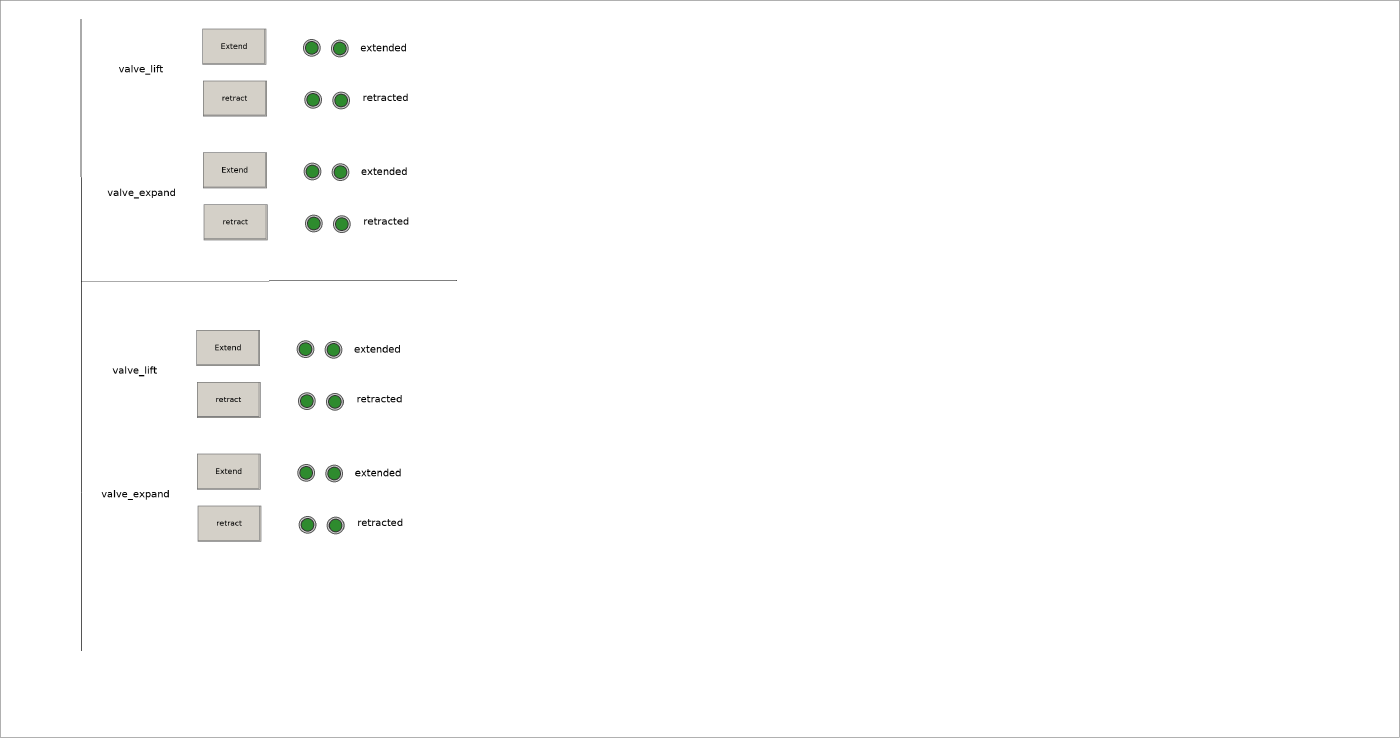
VISUALIZATION v_IO_fixtureClamp  // 2048x1080
    Line (118,28) (119,952)
    Label (126,88 160x26), "valve_lift"
    Button (296,42 93x52), "Extend", colour toggle: G_IO.arDO[55].Ch[10]
        OnMouseDown: execute { G_IO.arDO[55].Ch[10] := TRUE; G_IO.arDO[55].Ch[11] := FALSE; }
    Button (297,118 93x52), "retract", colour toggle: G_IO.arDO[55].Ch[11]
        OnMouseDown: execute { G_IO.arDO[55].Ch[10] := FALSE; G_IO.arDO[55].Ch[11] := TRUE; }
    Lamp1 (441,55 30x30), variable: G_IO.arDI[77].Ch[0], style: Lamp-Lamp1-Green
    Lamp1 (443,131 30x30), variable: G_IO.arDI[77].Ch[1], style: Lamp-Lamp1-Green
    Label (495,57 132x26), "extended"
    Label (498,130 132x26), "retracted"
    Lamp1 (482,56 30x30), variable: G_IO.arDI[77].Ch[2], style: Lamp-Lamp1-Green
    Lamp1 (484,132 30x30), variable: G_IO.arDI[77].Ch[3], style: Lamp-Lamp1-Green
    Label (127,269 160x26), "valve_expand"
    Button (297,223 93x52), "Extend", colour toggle: G_IO.arDO[55].Ch[12]
        OnMouseDown: execute { G_IO.arDO[55].Ch[12] := TRUE; G_IO.arDO[55].Ch[13] := FALSE; }
    Button (298,299 93x52), "retract", colour toggle: G_IO.arDO[55].Ch[13]
        OnMouseDown: execute { G_IO.arDO[55].Ch[12] := FALSE; G_IO.arDO[55].Ch[13] := TRUE; }
    Lamp1 (442,236 30x30), variable: G_IO.arDI[77].Ch[4], style: Lamp-Lamp1-Green
    Lamp1 (444,312 30x30), variable: G_IO.arDI[77].Ch[5], style: Lamp-Lamp1-Green
    Label (496,238 132x26), "extended"
    Label (499,311 132x26), "retracted"
    Lamp1 (483,237 30x30), variable: G_IO.arDI[77].Ch[6], style: Lamp-Lamp1-Green
    Lamp1 (485,313 30x30), variable: G_IO.arDI[77].Ch[7], style: Lamp-Lamp1-Green
    Label (117,529 160x26), "valve_lift"
    Button (287,483 93x52), "Extend", colour toggle: G_IO.arDO[59].Ch[10]
        OnMouseDown: execute { G_IO.arDO[59].Ch[10] := TRUE; G_IO.arDO[59].Ch[11] := FALSE; }
    Button (288,559 93x52), "retract", colour toggle: G_IO.arDO[59].Ch[11]
        OnMouseDown: execute { G_IO.arDO[59].Ch[10] := FALSE; G_IO.arDO[59].Ch[11] := TRUE; }
    Lamp1 (432,496 30x30), variable: G_IO.arDI[78].Ch[0], style: Lamp-Lamp1-Green
    Lamp1 (434,572 30x30), variable: G_IO.arDI[78].Ch[1], style: Lamp-Lamp1-Green
    Label (486,498 132x26), "extended"
    Label (489,571 132x26), "retracted"
    Lamp1 (473,497 30x30), variable: G_IO.arDI[78].Ch[2], style: Lamp-Lamp1-Green
    Lamp1 (475,573 30x30), variable: G_IO.arDI[78].Ch[3], style: Lamp-Lamp1-Green
    Label (118,710 160x26), "valve_expand"
    Button (288,664 93x52), "Extend", colour toggle: G_IO.arDO[59].Ch[12]
        OnMouseDown: execute { G_IO.arDO[59].Ch[12] := TRUE; G_IO.arDO[59].Ch[13] := FALSE; }
    Button (289,740 93x52), "retract", colour toggle: G_IO.arDO[59].Ch[13]
        OnMouseDown: execute { G_IO.arDO[59].Ch[12] := FALSE; G_IO.arDO[59].Ch[13] := TRUE; }
    Lamp1 (433,677 30x30), variable: G_IO.arDI[78].Ch[4], style: Lamp-Lamp1-Green
    Lamp1 (435,753 30x30), variable: G_IO.arDI[78].Ch[5], style: Lamp-Lamp1-Green
    Label (487,679 132x26), "extended"
    Label (490,752 132x26), "retracted"
    Lamp1 (474,678 30x30), variable: G_IO.arDI[78].Ch[6], style: Lamp-Lamp1-Green
    Lamp1 (476,754 30x30), variable: G_IO.arDI[78].Ch[7], style: Lamp-Lamp1-Green
    Line (119,411) (668,410)
END_VISUALIZATION

(* stored: Version 1.1.0.1, ProductVersion 3.1.4024.12
   Visu v_IO_fixtureClamp: Id {2d168dd3-53ad-44d8-9a51-41df90e0f811} *)
